FUNCTION_BLOCK differential_protection_1 (* Composite Function Block Type *)
  (* Standard: 61499-2 *)
  (* Version 0.0, 3/23/2016, gulzha, nxtControl GmbH, template *)
  PACKAGE Main;
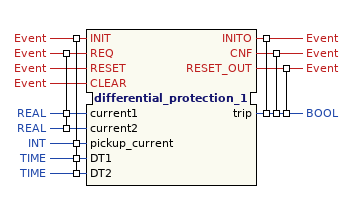
  EVENT_INPUT
    INIT WITH DT1, DT2, pickup_current; (* Initialization Request *)
    REQ WITH current1, current2; (* Normal Execution Request *)
    RESET;
    CLEAR;
  END_EVENT
  EVENT_OUTPUT
    INITO WITH trip; (* Initialization Confirm *)
    CNF WITH trip; (* Execution Confirmation *)
    RESET_OUT WITH trip;
  END_EVENT
  VAR_INPUT
    current1 : REAL;
    current2 : REAL;
    pickup_current : INT;
    DT1 : TIME; (* Delay Time *)
    DT2 : TIME; (* Delay Time *)
  END_VAR
  VAR_OUTPUT
    trip : BOOL;
  END_VAR
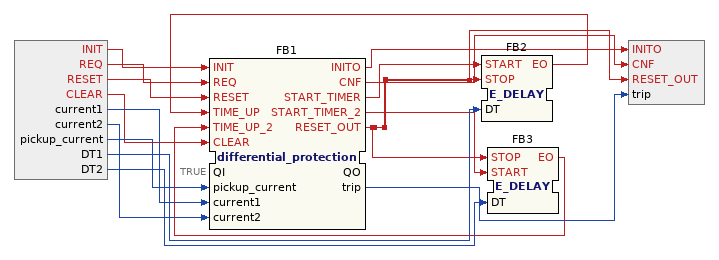
  FBS
    FB2 : E_DELAY;
    FB3 : E_DELAY;
    FB1 : differential_protection(QI := TRUE);
  END_FBS
  EVENT_CONNECTIONS
    INIT TO FB1.INIT;
    FB1.INITO TO INITO;
    FB1.CNF TO CNF;
    REQ TO FB1.REQ;
    RESET TO FB1.RESET;
    FB1.START_TIMER TO FB2.START;
    FB1.RESET_OUT TO FB2.STOP;
    FB1.RESET_OUT TO FB3.STOP;
    FB1.START_TIMER_2 TO FB3.START;
    FB1.RESET_OUT TO RESET_OUT;
    FB2.EO TO FB1.TIME_UP;
    FB3.EO TO FB1.TIME_UP_2;
    CLEAR TO FB1.CLEAR;
  END_CONNECTIONS
  DATA_CONNECTIONS
    DT1 TO FB2.DT;
    DT2 TO FB3.DT;
    FB1.trip TO trip;
    pickup_current TO FB1.pickup_current;
    current1 TO FB1.current1;
    current2 TO FB1.current2;
  END_CONNECTIONS
END_FUNCTION_BLOCK
